// TwinCAT 3 PLC project Test_Proj
// ProgramVersion: 3.1.4026.13
// libraries:
//   Tc2_Standard, * (Beckhoff Automation GmbH)
//   Tc2_System, * (Beckhoff Automation GmbH)
// project tree:
//   / PlcTask.TcTTO
//   POUs/ MAIN.TcPOU
//   Tests/ TestSuiteGVL.TcGVL, XtsCaGroupTestSuite.TcPOU, XtsHardwareTesting.TcPOU, XtsMoverTestSuite.TcPOU, XtsRunnerTesting.TcPOU, XtsTrackStub.TcPOU
// real-time tasks:
//   TASK PlcTask: cycle T#10ms, priority 20, ADS port 350

CONFIGURATION Test_Proj
    RESOURCE PLC ON TwinCAT3
        TASK PlcTask(INTERVAL := T#10ms, PRIORITY := 20);
        PROGRAM MAIN WITH PlcTask : MAIN;
    END_RESOURCE
END_CONFIGURATION

// ---- Tests/TestSuiteGVL.TcGVL
{attribute 'qualified_only'}
VAR_GLOBAL
	fbTestsuites:			FB_Testsuites;	
END_VAR

// ---- POUs/MAIN.TcPOU
PROGRAM MAIN
VAR
END_VAR

END_PROGRAM

// ---- Tests/XtsCaGroupTestSuite.TcPOU
FUNCTION_BLOCK XtsCaGroupTestSuite EXTENDS CollisionGroup
VAR
	fbTestSuites : FB_Testsuites;
	fbTestSuite : FB_Testsuite;
END_VAR

fbTestSuite();

CASE fbTestSuite.P_Testcase OF
	E_Testcase.Start:
		THIS^._ICaGroup := 1;
		fbTestSuite.P_Assert.M_Equals_DINT(1, THIS^.Cycle(), 'Cycle method did not return a complete');
		fbTestSuite.M_Testcase('GivenTheGroupExistsWhenCycleCalledThenCyclicTaskShouldRun',T#1S,'','',1);
		
	1:
		THIS^._ICaGroup := 0;
		fbTestSuite.P_Assert.M_Equals_DINT(-1, THIS^.Cycle(), 'Cycle method ran without vaild NC connection');
		fbTestSuite.M_Testcase('GivenNoCaRefWhenCycleCalledThenCyclicShouldNotRun',T#1S,'','',E_Testcase.Done);	
		
	E_Testcase.Done:;	 
END_CASE

METHOD FB_init : BOOL
VAR_INPUT
	bInitRetains : BOOL; // if TRUE, the retain variables are initialized (warm start / cold start)
	bInCopyCode : BOOL;  // if TRUE, the instance afterwards gets moved into the copy code (online change)
	XtsRunner : I_ObjectRunner;
END_VAR
//// Add Testsuite to Testsuites
TestSuiteGVL.fbTestsuites.M_Add(fbTestsuite);
TestSuiteGVL.fbTestsuites.P_Options.sFilePathName:= 'C:\test\report.xml';
END_METHOD

END_FUNCTION_BLOCK

// ---- Tests/XtsHardwareTesting.TcPOU
FUNCTION_BLOCK XtsHardwareTesting EXTENDS XTSHardware_V2
VAR
	bExecute:		BOOL;
	fbTestsuites:	FB_Testsuites;				// Testsuites
	XtsHardwareTestSuite : FB_Testsuite;
	
	// Test-vars	

END_VAR

// Run
fbTestsuites();

IF bExecute THEN
	// manual execute | override file path
	fbTestsuites.P_Options.sFilePathName:= 'C:\XtsHardwareTestReport.xml';
	bExecute:= NOT fbTestsuites.M_Request(E_Base.Execute);
END_IF

// Add Testsuite to Testsuites
fbTestsuites.M_Add(XtsHardwareTestSuite);

{region "XtsRunnerTestSuite"}
XtsHardwareTestSuite();
CASE XtsHardwareTestSuite.P_Testcase OF
//	E_Testcase.Start:
//		FOR i := 1 TO SystemParameters.nModuleNumber DO
//			f24V[i] := 0;	 
//		END_FOR
//		XtsHardwareTestSuite.P_Assert.M_Equals_DINT(1,THIS^.Is24VdcOK(),'check the 24vdc reports low correctly');
//		XtsHardwareTestSuite.M_Testcase('XtsHardware',T#1S,'','',1);
//	1:
//		FOR i := 1 TO SystemParameters.nModuleNumber DO
//			f24V[i] := 24000;	 
//		END_FOR 
//		f24V[2] := 18000;
//		XtsHardwareTestSuite.P_Assert.M_Equals_DINT(1,THIS^.Is24VOK(),'check the 24vdc reports low correctly with single sensor');
//		XtsHardwareTestSuite.M_Testcase('XtsHardware',T#1S,'','',2);
//	2:
//		XtsHardwareTestSuite.P_Assert.M_Equals_DINT(1,THIS^.Is48VOK(),'check the 24vdc reports 24vdcok correctly');
//		XtsHardwareTestSuite.M_Testcase('XtsHardware',T#1S,'','',E_Testcase.Done);

	E_Testcase.Done:;
		 
END_CASE
{endregion}

END_FUNCTION_BLOCK

// ---- Tests/XtsMoverTestSuite.TcPOU
FUNCTION_BLOCK XtsMoverTestSuite EXTENDS XtsMoverAxis
VAR
	fbTestSuite : FB_Testsuite;
	xtsTrack : XtsTrackStub;
	iXtsTrackStub : I_XtsTrack := xtsTrack;
	GearMasterFake : AXIS_REF;
END_VAR

fbTestSuite();

CASE fbTestSuite.P_Testcase OF
	E_Testcase.Start:
		THIS^._MyNCData.AxisId := 1;
		fbTestSuite.P_Assert.M_Equals_DINT(1, THIS^.Cycle(), 'Cycle method did not return a complete');
		fbTestSuite.M_Testcase('GivenTheMoverIsFoundWhenCycleCalledThenCyclicTaskShouldRun',T#1S,'','',1);
		
	1:
		THIS^._MyNCData.AxisId := 0;
		fbTestSuite.P_Assert.M_Equals_DINT(-1, THIS^.Cycle(), 'Cycle method ran without vaild NC connection');
		fbTestSuite.M_Testcase('GivenNoNCWhenCycleCalledThenCyclicShouldNotRun',T#1S,'','',2);	
		
	2:
		THIS^._CurrentTrack := 1; 
		_MyAxisStatus.Disabled := TRUE;
		fbTestSuite.P_Assert.M_Equals_DINT(1, THIS^.EnableMover(), 'Enable command failed when mover disabled');
		fbTestSuite.M_Testcase('GivenMoverDisabledWhenEnableCommandThenMoverEnables',T#1S,'','',3);
		
	3:
		_MyAxisStatus.Disabled := FALSE;
		fbTestSuite.P_Assert.M_Equals_DINT(-1, THIS^.EnableMover(), 'Enable Command was accepted when enabled');
		fbTestSuite.M_Testcase('GivenMoverEnabledWhenEnableComandThenEnableRejected',T#1S,'','',4);
		
	4:
		_MyAxisStatus.Disabled := FALSE;
		fbTestSuite.P_Assert.M_Equals_DINT(1, THIS^.DisableMover(), 'Disable command failed when mover was enabled');
		fbTestSuite.M_Testcase('GivenMoverEnabledWhenDisabledCommandMadeThenMoverDisables',T#1S,'','',5);
		
	5:	
		_MyAxisStatus.Disabled := TRUE;
		fbTestSuite.P_Assert.M_Equals_DINT(-1, THIS^.DisableMover(), 'Disable command accepted when mover was disabled');
		fbTestSuite.M_Testcase('GivenMoverDisabledWhenDisabledCommandMadeThenDisableRejected',T#1S,'','',6);
		
	6:
		_ActiveTrackLength := 5000.0;
		THIS^.Gap := 100.0;
		fbTestSuite.P_Assert.M_Equals_DINT(1,THIS^.MoveTo(RequiredPosition := 1000.0, MoveVelocity := 1000.0), 'Move command was rejected when mover was ready');
		fbTestSuite.M_Testcase('GivenMoverReadyWhenMoveCommandMadeThenMoverShouldAcceptMove',T#1S,'','',7);
		
	7:
		fbTestSuite.P_Assert.M_Equals_DINT(-1,THIS^.MoveTo(RequiredPosition := 1000.0, MoveVelocity := 5000.0), 'Move command was accepted when velocity too high');
		fbTestSuite.M_Testcase('WhenMoveCommandVelocityTooHighThenMoverShouldRejectMove',T#1S,'','',8);
		
	8: 
		_ActiveTrackLength := 1500.0;
		fbTestSuite.P_Assert.M_Equals_DINT(-1,THIS^.MoveTo(RequiredPosition := 2000.0, MoveVelocity := 1000.0), 'Move command was accepted when position outside modulo');
		fbTestSuite.M_Testcase('WhenMoveCommandOutsideModuloThenMoverShouldRejectMove',T#1S,'','',9);
		
	9:
		THIS^._MyAxisStatus.NotMoving := FALSE;
		fbTestSuite.P_Assert.M_Equals_DINT(1,THIS^.HaltAxis(),'Mover halt was rejected when mover moving');
		fbTestSuite.M_Testcase('GivenMovingMoverWhenHaltCommandThenMoverShouldAcceptHalt',T#1S,'','',10);
		
	10:
		THIS^._MyAxisStatus.NotMoving := FALSE;
		THIS^.HaltAxis();
		fbTestSuite.P_Assert.M_Equals_DINT(-1,THIS^.HaltAxis(), 'Mover halt was accepted when halt already commanded');
		fbTestSuite.M_Testcase('GivenHaltingMoverWhenHaltCommandGivenThenMoverShouldRejectCommand',T#1S,'','',11);
	
	11:
		THIS^.MoverHaltCommand.Abort();
		THIS^._MyAxisStatus.NotMoving := TRUE;
		fbTestSuite.P_Assert.M_Equals_DINT(-1,THIS^.HaltAxis(), 'Mover halt was accepted when velo was zero');
		fbTestSuite.M_Testcase('GivenStationaryMoverWhenHaltCommandedThenMoverShourlRejectCommand',T#1S,'','',12);
	
	12:
		THIS^.MoverResetCommand.Abort();
		THIS^._MyAxisStatus.Error := TRUE;
		fbTestSuite.P_Assert.M_Equals_DINT(1,THIS^.ResetAxis(), 'Mover reset was rejected when mover in error');
		fbTestSuite.M_Testcase('GivenMoverErrorWhenResetCommandedThemMoverShouldAcceptReset',T#1S,'','',13);
		
	13:
		THIS^._MyAxisStatus.Error := TRUE;
		THIS^.ResetAxis();
		fbTestSuite.P_Assert.M_Equals_DINT(-1,THIS^.ResetAxis(), 'Mover reset was accepted when reset already commanded');
		fbTestSuite.M_Testcase('GivenResettingMoverWhenResetCommandedThenMoverShouldRejectCommand',T#1S,'','',14);
		
	14:
		THIS^.MoverResetCommand.Abort();
		THIS^._MyAxisStatus.Error := FALSE;
		fbTestSuite.P_Assert.M_Equals_DINT(-1,THIS^.ResetAxis(), 'Mover reset was accepted when no error');
		fbTestSuite.M_Testcase('GivenOKMoverWhenResetCommandedThenMoverShouldRejectCommand',T#1S,'','',15);
		
	15:
		_MyAxisStatus.NotMoving := TRUE;
		fbTestSuite.P_Assert.M_Equals_DINT(1, THIS^.ActivateTrack(newTrack := 16#1,iXtsTrackStub), 'Mover rejected valid active track command');
		fbTestSuite.M_Testcase('GivenAStationaryMoverWhenActiveTrackGivenThenMoverShouldAcceptNewTrack',T#1S,'','',16);
		
	16:
		THIS^.MoverActivateTrackCommand.Abort();
		_MyAxisStatus.NotMoving := FALSE;
		fbTestSuite.P_Assert.M_Equals_DINT(-1,THIS^.ActivateTrack(newTrack := 16#1,iXtsTrackStub), 'Mover accepted track command when moving');
		fbTestSuite.M_Testcase('GivenMovingMoverWhenActiveTrackCommandThenMoverSouldRejectCommand',T#1S,'','',17);
		
	17:
		THIS^.MoverActivateTrackCommand.Abort();
		fbTestSuite.P_Assert.M_Equals_DINT(-1, THIS^.ActivateTrack(newTrack := 16#1,iXtsTrackStub), 'Mover Accepted invalid track');
		fbTestSuite.M_Testcase('GivenInvalidTrackWhenActiveTrackCommandThenMoverShouldReject',T#1S,'','',18);
		
	18:
		THIS^._CurrentTrack := 0; 
		fbTestSuite.P_Assert.M_Equals_DINT(-1, THIS^.EnableMover(), 'Mover accepted enable without a valid track');
		fbTestSuite.M_Testcase('GivenNoTracksRegisteredWhenEnebleGivenThenMoverShouldReject',T#1S,'','',19);
		
	19: 
		THIS^.MoverActivateTrackCommand.Abort();
		_MyAxisStatus.NotMoving := TRUE;
		fbTestSuite.P_Assert.M_Equals_DINT(1, THIS^.ActivateTrack(NewTrack := 1, Track := iXtsTrackStub), 'Mover did not set the track length when given new track');
		fbTestSuite.M_Testcase('GivenNewTrackWhenActivateTrackCalledThenMoverShouldAcceptNewTrackLength',T#1S,'','',20);
		
	20:
		THIS^.MyMasterRef REF= 0;
		_ActiveTrackLength := 2500.0;
		THIS^.axesGear.Abort();
		fbTestSuite.P_Assert.M_Equals_DINT(-1,THIS^.Gear(1000.0,2000.0), 'Mover accepted command with no valid master');
		fbTestSuite.M_Testcase('GivenNoMasterWhenGearCommandThenMoverShouldReject',T#1S,'','',21);
		
	21:
		THIS^.axesGear.Abort();
		THIS^.MyMasterRef REF= GearMasterFake;
		_ActiveTrackLength := 2500.0;
		fbTestSuite.P_Assert.M_Equals_DINT(1, THIS^.Gear(1000.0,2000.0), 'The Mover rejected valid gear command');
		fbTestSuite.M_Testcase('GivenAValidMoverWhenGearCommandIssuedThenMoverShouldAcceptCommand',T#1S,'','',22);
		
	22:
		THIS^.MyMasterRef REF= GearMasterFake;
		THIS^.axesGear.Abort();
		_ActiveTrackLength := 4000.0;
		fbTestSuite.P_Assert.M_Equals_DINT(-1,THIS^.Gear(5000.0,1000.0), 'Mover accepted master position outside track');
		fbTestSuite.M_Testcase('GivenAValidMoverWhenGearCommandOutsideTrackThenMoverShouldReject',T#1S,'','',23);
		
	23:
		THIS^.MyMasterRef REF= GearMasterFake;
		THIS^.axesGear.Abort();
		_ActiveTrackLength := 5000.0;
		fbTestSuite.P_Assert.M_Equals_DINT(-1,THIS^.Gear(2000.0,10000.0), 'Mover accepted slave position outside track');
		fbTestSuite.M_Testcase('GivenAValidMoverWhenGearCommandOutsideTrackThenMoverShouldReject',T#1S,'','',E_Testcase.Done);
		
	E_Testcase.Done:;	 
END_CASE

METHOD FB_init : BOOL
VAR_INPUT
	bInitRetains : BOOL; // if TRUE, the retain variables are initialized (warm start / cold start)
	bInCopyCode : BOOL;  // if TRUE, the instance afterwards gets moved into the copy code (online change)
	XtsRunner : I_ObjectRunner;
END_VAR
//// Add Testsuite to Testsuites
TestSuiteGVL.fbTestsuites.M_Add(fbTestsuite);
TestSuiteGVL.fbTestsuites.P_Options.sFilePathName:= 'C:\test\report.xml';
END_METHOD

END_FUNCTION_BLOCK

// ---- Tests/XtsTrackStub.TcPOU
FUNCTION_BLOCK XtsTrackStub IMPLEMENTS I_XtsTrack
VAR_INPUT
END_VAR
VAR_OUTPUT
END_VAR
VAR
	_trackLength : MC_LREAL  := 1000;
END_VAR

{warning 'add property implementation'}
PROPERTY MyOTCID : OTCID
GET
END_GET
SET
END_SET
END_PROPERTY

{warning 'add property implementation'}
PROPERTY TrackLength : MC_Lreal
GET
tracklength := _trackLength;
END_GET
END_PROPERTY

END_FUNCTION_BLOCK

// ---- Tests/XtsRunnerTesting.TcPOU
FUNCTION_BLOCK XtsRunnerTesting EXTENDS ObjectRunner
VAR
	XtsRunnerTestSuite : FB_Testsuite;
	
	// Test-vars	
	arrCyclicModules : ARRAY[1..101] OF XtsMoverAxis(THIS^);
	//InitialiseModule : XTSHardware_V2(THIS^);
	InitAddedCheck : BOOL;
	CyclicAddedCheck: BOOL;
END_VAR

{region "XtsRunnerTestSuite"}
XtsRunnerTestSuite();
CASE XtsRunnerTestSuite.P_Testcase OF
	E_Testcase.Start:
		XtsRunnerTestSuite.M_Testcase('XtsRunner',T#1S,'','',1);
			 
	1:
		XtsRunnerTestSuite.P_Assert.M_Equals_INT(0,THIS^.GetModuleCount(),'check modules empty');
		THIS^.ModuleCount := 1;
		XtsRunnerTestSuite.P_Assert.M_Equals_INT(1,THIS^.GetModuleCount(),'check module count seen correctly');
		THIS^.ModuleCount := 0;
		XtsRunnerTestSuite.M_Testcase('XtsRunner',T#1S,'','',2);
		 
	2:
		XtsRunnerTestSuite.P_Assert.M_Equals_DINT(2,THIS^.AddComponent(arrCyclicModules[1]),'Try register 1 cyclic module');
		CyclicAddedCheck := THIS^.CyclicModules[0] <> 0;	 
		XtsRunnerTestSuite.P_Assert.M_IsTRUE(CyclicAddedCheck,'module not added in array correctly'); 
		XtsRunnerTestSuite.M_Testcase('XtsRunner',T#1S,'','',3);
		THIS^.CyclicModules[0] := 0;
		THIS^.ModuleCount := 0;	 
		CyclicAddedCheck := FALSE;
			 
	3: 
		XtsRunnerTestSuite.P_Assert.M_Equals_DINT(2,THIS^.AddComponent(arrCyclicModules[1]),'Try register 1 cyclic module');
		InitAddedCheck := NOT (THIS^.InitialiseModules[0] <> 0);
		XtsRunnerTestSuite.P_Assert.M_IsTRUE(InitAddedCheck,'Initial interface added incorrectly');
		XtsRunnerTestSuite.M_Testcase('XtsRunner',T#1S,'','',4);
		THIS^.CyclicModules[0] := 0;
		THIS^.ModuleCount := 0;	 
		InitAddedCheck := FALSE;
	 
	4:
		XtsRunnerTestSuite.P_Assert.M_Equals_INT(0,THIS^.GetModuleCount(),'check modules empty');
		FOR i := 1 TO 100 DO 
			THIS^.AddComponent(arrCyclicModules[i]);
		END_FOR
		XtsRunnerTestSuite.P_Assert.M_Equals_DINT(1,THIS^.AddComponent(arrCyclicModules[101]),'add to many modules should be rejected');
		XtsRunnerTestSuite.M_Testcase('XtsRunner',T#1S,'','',5);
		FOR i := 0 TO 99 DO 
			THIS^.CyclicModules[i] := 0;
		END_FOR
		THIS^.ModuleCount := 0;		 
	
	5:
		THIS^.Clear();
		XtsRunnerTestSuite.P_Assert.M_Equals_DINT(2,THIS^.AddComponent(arrCyclicModules[1]),'try register a single cyclic modulea');
		XtsRunnerTestSuite.P_Assert.M_Equals_INT(1,THIS^.GetModuleCount(),'check module added in count'); 
		XtsRunnerTestSuite.P_Assert.M_Equals_DINT(2,THIS^.RemoveModule(arrCyclicModules[1]),'remove the same module from module list');
		XtsRunnerTestSuite.P_Assert.M_Equals_INT(0,THIS^.GetModuleCount(),'check modules empty');	 
		XtsRunnerTestSuite.M_Testcase('XtsRunner',T#1S,'','',6);
	
	6:
		XtsRunnerTestSuite.P_Assert.M_Equals_INT(0,THIS^.GetModuleCount(),'check modules empty');
		XtsRunnerTestSuite.P_Assert.M_Equals_DINT(1,THIS^.RemoveModule(arrCyclicModules[1]),'Try remove from empty module list');	 
		XtsRunnerTestSuite.P_Assert.M_Equals_INT(0,THIS^.GetModuleCount(),'check modules empty big check');
		XtsRunnerTestSuite.M_Testcase('XtsRunner',T#1S,'','',7);
		
//	7:
//		THIS^.AddComponent(InitialiseModule);
//		CyclicAddedCheck := THIS^.CyclicModules[0] <> 0;	
//		InitAddedCheck := THIS^.InitialiseModules[0] <> 0;
//		XtsRunnerTestSuite.P_Assert.M_IsTRUE(CyclicAddedCheck,'module not added in array correctly');
//		XtsRunnerTestSuite.P_Assert.M_IsTRUE(InitAddedCheck,'Initial interface not added correctly'); 
//		XtsRunnerTestSuite.M_Testcase('XtsRunner',T#1S,'','',8);
//		THIS^.CyclicModules[0] := 0;
//		THIS^.InitialiseModules[0] := 0;
//		THIS^.ModuleCount := 0;
//		THIS^.InitModuleCount := 0;	 
			 
//	8:
//		THIS^.AddComponent(InitialiseModule);
//		XtsRunnerTestSuite.P_Assert.M_Equals_INT(1,THIS^.InitModuleCount,'initialisation module not been counted correctly');	
//		XtsRunnerTestSuite.M_Testcase('XtsRunner',T#1S,'','',9);
//		THIS^.CyclicModules[0] := 0;
//		THIS^.InitialiseModules[0] := 0;
//		THIS^.CyclicModules[0] := 0;
//		THIS^.InitialiseModules[0] := 0;
//		THIS^.ModuleCount := 0;
//		THIS^.InitModuleCount := 0; 
			 
//	9:
//		THIS^.AddComponent(InitialiseModule);
//		XtsRunnerTestSuite.P_Assert.M_Equals_INT(1,THIS^.InitModuleCount,'initialisation module not been counted correctly');
//		THIS^.RemoveModule(InitialiseModule);
//		XtsRunnerTestSuite.P_Assert.M_Equals_INT(0,THIS^.InitModuleCount,'initialisation module not been removed correctly');
//		XtsRunnerTestSuite.M_Testcase('XtsRunner',T#1S,'','',10);
//		THIS^.CyclicModules[0] := 0;
//		THIS^.InitialiseModules[0] := 0;
//		THIS^.CyclicModules[0] := 0;
//		THIS^.InitialiseModules[0] := 0;
//		THIS^.ModuleCount := 0;
//		THIS^.InitModuleCount := 0;
		
	10:
		THIS^.Clear();
		XtsRunnerTestSuite.M_Testcase('XtsRunner',T#1S,'','',E_Testcase.Done);
	E_Testcase.Done:;	 
END_CASE
{endregion}

METHOD FB_init : BOOL
VAR_INPUT
	bInitRetains : BOOL; // if TRUE, the retain variables are initialized (warm start / cold start)
	bInCopyCode : BOOL;  // if TRUE, the instance afterwards gets moved into the copy code (online change)
END_VAR
//// Add Testsuite to Testsuites
TestSuiteGVL.fbTestsuites.M_Add(XtsRunnerTestSuite);
TestSuiteGVL.fbTestsuites.P_Options.sFilePathName:= 'C:\test\report.xml';
END_METHOD

END_FUNCTION_BLOCK
